// TIA Portal project "MANIPULATOR_Planinc_Novak(V9)_KONCNA" (V15.1)

(* hardware
DEVICE "S7-1200 station_1"  S7-1200 Station
   slot 0: "Rack_0"  S7-1200 Rack  Rack  V1.0
   slot 1: "PLC_1"  CPU 1214C DC/DC/DC  6ES7 214-1AG40-0XB0  V4.2
      slot 3: "DI 4x24VDC_1"  DI4 signal board (200 kHz)  6ES7 221-3BD30-0XB0  V1.0
   slot 2: "DI 8/DQ 8x24VDC_1"  SM 1223 DI8/DQ8 x 24VDC  6ES7 223-1BH30-0XB0  V1.0
   slot 3: "DI 8/DQ 8x24VDC_2"  6ES7 223-1BH32-0XB0  V2.0
*)

// ===== PLC "PLC_1"  CPU 1214C DC/DC/DC =====

VAR_GLOBAL   // PLC tag table "Default tag table"
   "START" AT %I0.0 : Bool;
   "STOP" AT %I0.1 : Bool;
   "AUTO/MAN" AT %I0.2 : Bool;
   "a0" AT %I0.3 : Bool;
   "a1" AT %I0.4 : Bool;
   "b0" AT %I12.7 : Bool;
   "b1" AT %I0.5 : Bool;
   "c1" AT %I0.6 : Bool;
   "k0" AT %I8.4 : Bool;
   "k1" AT %I8.5 : Bool;
   "j0" AT %I8.2 : Bool;
   "j1" AT %I8.3 : Bool;
   "i1" AT %I8.1 : Bool;
   "i0" AT %I8.0 : Bool;
   "e1" AT %I1.0 : Bool;
   "e0" AT %I0.7 : Bool;
   "e2" AT %I1.1 : Bool;
   "h0" AT %I1.4 : Bool;
   "h1" AT %I1.5 : Bool;
   "g0" AT %I1.2 : Bool;
   "g1" AT %I1.3 : Bool;
   "dp3" AT %I12.5 : Bool;
   "A" AT %Q0.0 : Bool;
   "B" AT %Q0.1 : Bool;
   "C" AT %Q0.2 : Bool;
   "D" AT %Q0.3 : Bool;
   "E+" AT %Q0.4 : Bool;
   "E-" AT %Q0.5 : Bool;
   "F+" AT %Q0.6 : Bool;
   "G+" AT %Q0.7 : Bool;
   "H+" AT %Q1.0 : Bool;
   "I+" AT %Q1.1 : Bool;
   "J+" AT %Q8.0 : Bool;
   "J-" AT %Q8.1 : Bool;
   "K+" AT %Q8.2 : Bool;
   "V+" AT %Q8.3 : Bool;
   "FM" AT %Q8.4 : Bool;
   "M(J)" AT %M0.0 : Bool;
   "M(E-)" AT %M0.1 : Bool;
   "PULZ" AT %M0.2 : Bool;
   "M(E+)" AT %M0.3 : Bool;
   "kor1" AT %M0.4 : Bool;
   "kor3" AT %M0.5 : Bool;
   "dp1" AT %I8.7 : Bool;
   "dp2" AT %I12.4 : Bool;
   "RS timer" AT %M0.7 : Bool;
   "kor2" AT %M0.6 : Bool;
   "kor4" AT %M1.0 : Bool;
   "kor4.1" AT %M1.1 : Bool;
   "kor5" AT %M1.2 : Bool;
   "kor5.1" AT %M1.3 : Bool;
   "kor5.2" AT %M1.4 : Bool;
   "kor 6" AT %M1.5 : Bool;
   "kor 6.1" AT %M1.6 : Bool;
   "kor 6.2" AT %M1.7 : Bool;
   "kor 6.3" AT %M2.0 : Bool;
   "kor 7" AT %M2.1 : Bool;
   "napaka" AT %M2.2 : Bool;
   "Tag_1" AT %M2.3 : Bool;
   "Tag_2" AT %M2.4 : Bool;
   "Tag_3" AT %M2.5 : Bool;
   "Tag_4" AT %M2.6 : Bool;
   "Tag_5" AT %M2.7 : Bool;
END_VAR

DATA_BLOCK "Data_block_1"   // DB1
{ S7_Optimized_Access := 'FALSE' }
VERSION : 0.1
   VAR
      check_ok : Bool;
      check_not_ok : Bool;
   END_VAR
BEGIN
END_DATA_BLOCK

// folder: System blocks/Program resources

DATA_BLOCK "T4.1"   // DB2
{ S7_Optimized_Access := 'TRUE' }
AUTHOR : Simatic
FAMILY : IEC
NAME : IEC_TMR
VERSION : 1.0
// stored: InstanceOfName IEC_TIMER
"IEC_TIMER"
BEGIN
END_DATA_BLOCK

DATA_BLOCK "stevec1"   // DB3
{ S7_Optimized_Access := 'TRUE' }
AUTHOR : Simatic
FAMILY : IEC
NAME : CNTR
VERSION : 1.0
// stored: InstanceOfName IEC_COUNTER
"IEC_COUNTER"
BEGIN
END_DATA_BLOCK

DATA_BLOCK "napaka 2"   // DB5
{ S7_Optimized_Access := 'TRUE' }
AUTHOR : Simatic
FAMILY : IEC
NAME : IEC_TMR
VERSION : 1.0
// stored: InstanceOfName IEC_TIMER
"IEC_TIMER"
BEGIN
END_DATA_BLOCK

// folder: (top level)

ORGANIZATION_BLOCK "Main"   // OB1, LAD, ProgramCycle
TITLE = "Main Program Sweep (Cycle)"
{ S7_Optimized_Access := 'TRUE' }
VERSION : 0.1
   VAR_INPUT
      Initial_Call : Bool;   // Initial call of this OB
      Remanence : Bool;   // =True, if remanent data are available
   END_VAR
   VAR_TEMP   // added for the SCL form of the ladder/FBD networks
      _w1 : Bool;
      _w2 : Bool;
   END_VAR
BEGIN

REGION Network 1: števec
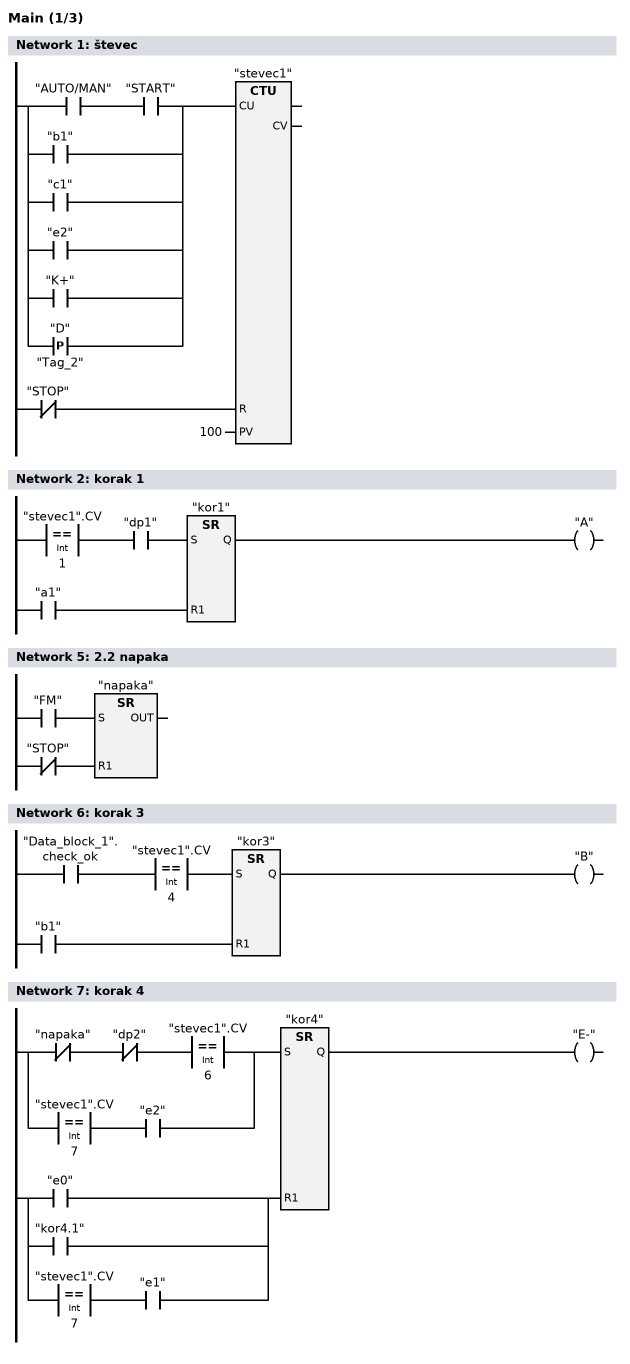
   #_w1 := "D" AND NOT "Tag_2";   // rising edge of "D"
   "Tag_2" := "D";
   "stevec1".CTU(CU := ("AUTO/MAN" AND "START") OR "b1" OR "c1" OR "e2" OR "K+" OR #_w1,
                 R := NOT "STOP",
                 PV := 100);
END_REGION

REGION Network 2: korak 1
   RUNG wire#powerrail
      { S7_Templates := "SrcType := Int" } EQ_Contact(in1 := "stevec1".CV, in2 := 1)
      Contact( "dp1" )
      S_SR(operand := "kor1", r1 := wire#w1)
      Coil( "A" )
   END_RUNG
   RUNG wire#powerrail
      Contact( "a1" )
   END_RUNG wire#w1
   // the same network as SCL:
   IF ("stevec1".CV = 1) AND "dp1" THEN
       "kor1" := TRUE;   // SR flip-flop
   END_IF;
   IF "a1" THEN "kor1" := FALSE; END_IF;
   "A" := "kor1";
END_REGION

REGION Network 3: korak 2
END_REGION

REGION Network 4: korak 2.1
END_REGION

REGION Network 5: 2.2 napaka
   RUNG wire#powerrail
      Contact( "FM" )
      S_SR(operand := "napaka", r1 := wire#w1)
   END_RUNG
   RUNG wire#powerrail
      I_Contact( "STOP" )
   END_RUNG wire#w1
   // the same network as SCL:
   IF "FM" THEN
       "napaka" := TRUE;   // SR flip-flop
   END_IF;
   IF NOT "STOP" THEN "napaka" := FALSE; END_IF;
END_REGION

REGION Network 6: korak 3
   RUNG wire#powerrail
      Contact( "Data_block_1".check_ok )
      { S7_Templates := "SrcType := Int" } EQ_Contact(in1 := "stevec1".CV, in2 := 4)
      S_SR(operand := "kor3", r1 := wire#w1)
      Coil( "B" )
   END_RUNG
   RUNG wire#powerrail
      Contact( "b1" )
   END_RUNG wire#w1
   // the same network as SCL:
   IF "Data_block_1".check_ok AND ("stevec1".CV = 4) THEN
       "kor3" := TRUE;   // SR flip-flop
   END_IF;
   IF "b1" THEN "kor3" := FALSE; END_IF;
   "B" := "kor3";
END_REGION

REGION Network 7: korak 4
   RUNG wire#powerrail
      I_Contact( "napaka" )
      I_Contact( "dp2" )
      { S7_Templates := "SrcType := Int" } EQ_Contact(in1 := "stevec1".CV, in2 := 6)
      wire#w1
      S_SR(operand := "kor4", r1 := wire#w2)
      Coil( "E-" )
   END_RUNG
   RUNG wire#powerrail
      { S7_Templates := "SrcType := Int" } EQ_Contact(in1 := "stevec1".CV, in2 := 7)
      Contact( "e2" )
   END_RUNG wire#w1
   RUNG wire#powerrail
      Contact( "e0" )
   END_RUNG wire#w2
   RUNG wire#powerrail
      Contact( "kor4.1" )
   END_RUNG wire#w2
   RUNG wire#powerrail
      { S7_Templates := "SrcType := Int" } EQ_Contact(in1 := "stevec1".CV, in2 := 7)
      Contact( "e1" )
   END_RUNG wire#w2
   // the same network as SCL:
   IF (NOT "napaka" AND NOT "dp2" AND ("stevec1".CV = 6)) OR (("stevec1".CV = 7) AND "e2") THEN
       "kor4" := TRUE;   // SR flip-flop
   END_IF;
   IF "e0" OR "kor4.1" OR (("stevec1".CV = 7) AND "e1") THEN "kor4" := FALSE; END_IF;
   "E-" := "kor4";
END_REGION

REGION Network 8: korak 4.1
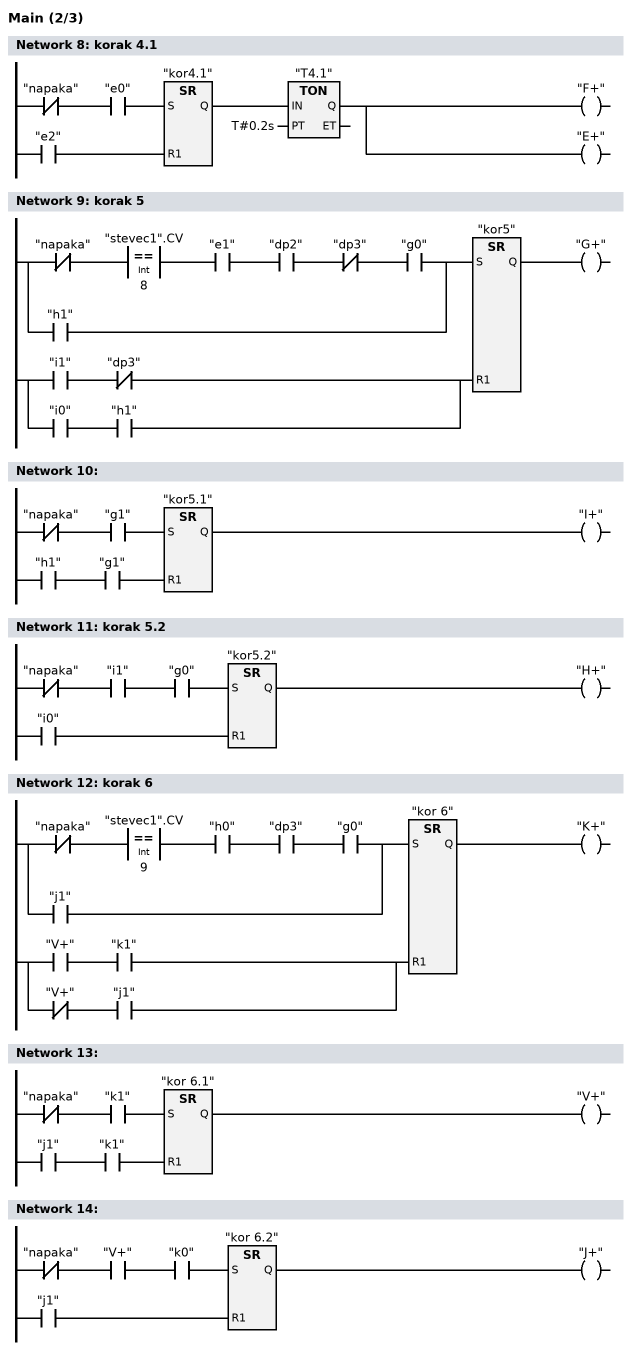
   IF NOT "napaka" AND "e0" THEN
       "kor4.1" := TRUE;   // SR flip-flop
   END_IF;
   IF "e2" THEN "kor4.1" := FALSE; END_IF;
   "T4.1".TON(IN := "kor4.1", PT := T#0.2s);
   "F+" := "T4.1".Q;
   "E+" := "T4.1".Q;
END_REGION

REGION Network 9: korak 5
   RUNG wire#powerrail
      I_Contact( "napaka" )
      { S7_Templates := "SrcType := Int" } EQ_Contact(in1 := "stevec1".CV, in2 := 8)
      Contact( "e1" )
      Contact( "dp2" )
      I_Contact( "dp3" )
      Contact( "g0" )
      wire#w1
      S_SR(operand := "kor5", r1 := wire#w2)
      Coil( "G+" )
   END_RUNG
   RUNG wire#powerrail
      Contact( "h1" )
   END_RUNG wire#w1
   RUNG wire#powerrail
      Contact( "i1" )
      I_Contact( "dp3" )
   END_RUNG wire#w2
   RUNG wire#powerrail
      Contact( "i0" )
      Contact( "h1" )
   END_RUNG wire#w2
   // the same network as SCL:
   IF (NOT "napaka" AND ("stevec1".CV = 8) AND "e1" AND "dp2" AND NOT "dp3" AND "g0") OR "h1" THEN
       "kor5" := TRUE;   // SR flip-flop
   END_IF;
   IF ("i1" AND NOT "dp3") OR ("i0" AND "h1") THEN "kor5" := FALSE; END_IF;
   "G+" := "kor5";
END_REGION

REGION Network 10
   RUNG wire#powerrail
      I_Contact( "napaka" )
      Contact( "g1" )
      S_SR(operand := "kor5.1", r1 := wire#w1)
      Coil( "I+" )
   END_RUNG
   RUNG wire#powerrail
      Contact( "h1" )
      Contact( "g1" )
   END_RUNG wire#w1
   // the same network as SCL:
   IF NOT "napaka" AND "g1" THEN
       "kor5.1" := TRUE;   // SR flip-flop
   END_IF;
   IF "h1" AND "g1" THEN "kor5.1" := FALSE; END_IF;
   "I+" := "kor5.1";
END_REGION

REGION Network 11: korak 5.2
   RUNG wire#powerrail
      I_Contact( "napaka" )
      Contact( "i1" )
      Contact( "g0" )
      S_SR(operand := "kor5.2", r1 := wire#w1)
      Coil( "H+" )
   END_RUNG
   RUNG wire#powerrail
      Contact( "i0" )
   END_RUNG wire#w1
   // the same network as SCL:
   IF NOT "napaka" AND "i1" AND "g0" THEN
       "kor5.2" := TRUE;   // SR flip-flop
   END_IF;
   IF "i0" THEN "kor5.2" := FALSE; END_IF;
   "H+" := "kor5.2";
END_REGION

REGION Network 12: korak 6
   RUNG wire#powerrail
      I_Contact( "napaka" )
      { S7_Templates := "SrcType := Int" } EQ_Contact(in1 := "stevec1".CV, in2 := 9)
      Contact( "h0" )
      Contact( "dp3" )
      Contact( "g0" )
      wire#w1
      S_SR(operand := "kor 6", r1 := wire#w2)
      Coil( "K+" )
   END_RUNG
   RUNG wire#powerrail
      Contact( "j1" )
   END_RUNG wire#w1
   RUNG wire#powerrail
      Contact( "V+" )
      Contact( "k1" )
   END_RUNG wire#w2
   RUNG wire#powerrail
      I_Contact( "V+" )
      Contact( "j1" )
   END_RUNG wire#w2
   // the same network as SCL:
   IF (NOT "napaka" AND ("stevec1".CV = 9) AND "h0" AND "dp3" AND "g0") OR "j1" THEN
       "kor 6" := TRUE;   // SR flip-flop
   END_IF;
   IF ("V+" AND "k1") OR (NOT "V+" AND "j1") THEN "kor 6" := FALSE; END_IF;
   "K+" := "kor 6";
END_REGION

REGION Network 13
   RUNG wire#powerrail
      I_Contact( "napaka" )
      Contact( "k1" )
      S_SR(operand := "kor 6.1", r1 := wire#w1)
      Coil( "V+" )
   END_RUNG
   RUNG wire#powerrail
      Contact( "j1" )
      Contact( "k1" )
   END_RUNG wire#w1
   // the same network as SCL:
   IF NOT "napaka" AND "k1" THEN
       "kor 6.1" := TRUE;   // SR flip-flop
   END_IF;
   IF "j1" AND "k1" THEN "kor 6.1" := FALSE; END_IF;
   "V+" := "kor 6.1";
END_REGION

REGION Network 14
   RUNG wire#powerrail
      I_Contact( "napaka" )
      Contact( "V+" )
      Contact( "k0" )
      S_SR(operand := "kor 6.2", r1 := wire#w1)
      Coil( "J+" )
   END_RUNG
   RUNG wire#powerrail
      Contact( "j1" )
   END_RUNG wire#w1
   // the same network as SCL:
   IF NOT "napaka" AND "V+" AND "k0" THEN
       "kor 6.2" := TRUE;   // SR flip-flop
   END_IF;
   IF "j1" THEN "kor 6.2" := FALSE; END_IF;
   "J+" := "kor 6.2";
END_REGION

REGION Network 15
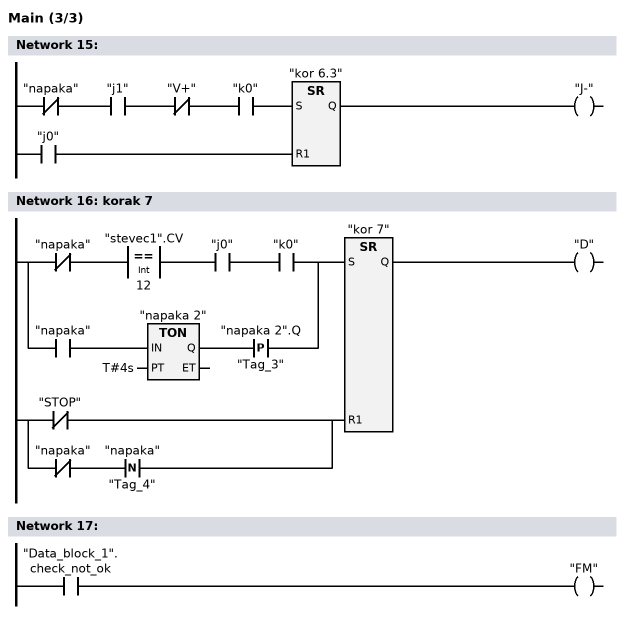
   RUNG wire#powerrail
      I_Contact( "napaka" )
      Contact( "j1" )
      I_Contact( "V+" )
      Contact( "k0" )
      S_SR(operand := "kor 6.3", r1 := wire#w1)
      Coil( "J-" )
   END_RUNG
   RUNG wire#powerrail
      Contact( "j0" )
   END_RUNG wire#w1
   // the same network as SCL:
   IF NOT "napaka" AND "j1" AND NOT "V+" AND "k0" THEN
       "kor 6.3" := TRUE;   // SR flip-flop
   END_IF;
   IF "j0" THEN "kor 6.3" := FALSE; END_IF;
   "J-" := "kor 6.3";
END_REGION

REGION Network 16: korak 7
   "napaka 2".TON(IN := "napaka", PT := T#4s);
   #_w1 := "napaka 2".Q AND "napaka 2".Q AND NOT "Tag_3";   // rising edge of "napaka 2".Q
   "Tag_3" := "napaka 2".Q;
   #_w2 := NOT "napaka" AND NOT "napaka" AND "Tag_4";   // falling edge of "napaka"
   "Tag_4" := "napaka";
   IF (NOT "napaka" AND ("stevec1".CV = 12) AND "j0" AND "k0") OR #_w1 THEN
       "kor 7" := TRUE;   // SR flip-flop
   END_IF;
   IF NOT "STOP" OR #_w2 THEN "kor 7" := FALSE; END_IF;
   "D" := "kor 7";
END_REGION

REGION Network 17
   RUNG wire#powerrail
      Contact( "Data_block_1".check_not_ok )
      Coil( "FM" )
   END_RUNG
   // the same network as SCL:
   "FM" := "Data_block_1".check_not_ok;
END_REGION
END_ORGANIZATION_BLOCK